// TIA Portal project "Assembler" (V16)
// Vorlageprojekt für das Buch mit Zielsystem S7-1200

(* hardware
DEVICE "S7-1200-Station_1"  S7-1200 Station
   slot 0: "Baugruppenträger_0"  Rack  V1.0
   slot 1: "PLC_1"  CPU 1211C DC/DC/DC  6ES7 211-1AE40-0XB0  V4.1
*)

// ===== PLC "PLC_1"  CPU 1211C DC/DC/DC =====

VAR_GLOBAL   // PLC tag table "Standard-Variablentabelle"
   "Start" AT %I0.0 : Bool;
   "Stop" AT %I0.1 : Bool;
   "Vision sensor (bool 0)" AT %I0.2 : Bool;
   "Vision sensor (bool 1)" AT %I0.3 : Bool;
   "pusher base (FL)" AT %I0.4 : Bool;
   "pusher base (BL)" AT %I0.5 : Bool;
   "pusher LID (FL)" AT %I0.6 : Bool;
   "pusher LID (BL)" AT %I0.7 : Bool;
   "DS BASE" AT %I1.0 : Bool;
   "DS LID" AT %I1.1 : Bool;
   "Base Clamped" AT %I1.2 : Bool;
   "LID Clamped" AT %I1.3 : Bool;
   "Item Leaving" AT %I1.4 : Bool;
   "Moving Z" AT %I1.5 : Bool;
   "Moving X" AT %I1.6 : Bool;
   "Item Detected" AT %I1.7 : Bool;
   "Sensor Base" AT %I2.0 : Bool;
   "Sensor LID" AT %I2.1 : Bool;
   "First Conv" AT %Q0.0 : Bool;
   "Main Conv" AT %Q0.1 : Bool;
   "Pusher Base" AT %Q0.2 : Bool;
   "Pusher LID" AT %Q0.3 : Bool;
   "Base Conv" AT %Q0.4 : Bool;
   "LID Conv" AT %Q0.5 : Bool;
   "Base Clamp" AT %Q0.6 : Bool;
   "LID Clamp" AT %Q0.7 : Bool;
   "Item Leave" AT %Q1.0 : Bool;
   "Move z" AT %Q1.1 : Bool;
   "Move x" AT %Q1.2 : Bool;
   "Grab" AT %Q1.3 : Bool;
   "X" AT %M0.0 : Bool;
   "X1" AT %M0.1 : Bool;
   "X2" AT %M0.2 : Bool;
   "X3" AT %M0.3 : Bool;
   "X4" AT %M0.4 : Bool;
   "X5" AT %M0.5 : Bool;
   "X6" AT %M0.6 : Bool;
   "X7" AT %M0.7 : Bool;
   "X8" AT %M1.0 : Bool;
   "X9" AT %M1.1 : Bool;
   "X10" AT %M1.2 : Bool;
   "X11" AT %M1.3 : Bool;
   "X12" AT %M1.4 : Bool;
   "X13" AT %M1.5 : Bool;
   "X14" AT %M1.6 : Bool;
   "X15" AT %M1.7 : Bool;
   "X16" AT %M2.0 : Bool;
   "X17" AT %M2.1 : Bool;
   "X18" AT %M2.2 : Bool;
   "X19" AT %M2.3 : Bool;
   "X20" AT %M2.4 : Bool;
   "X21" AT %M3.0 : Bool;
END_VAR

// folder: System blocks/Program resources

DATA_BLOCK "C1"   // DB1
{ S7_Optimized_Access := 'TRUE' }
AUTHOR : Simatic
FAMILY : IEC
NAME : CNTR
VERSION : 1.0
// stored: InstanceOfName IEC_COUNTER
"IEC_COUNTER"
BEGIN
END_DATA_BLOCK

DATA_BLOCK "T1"   // DB2
{ S7_Optimized_Access := 'TRUE' }
AUTHOR : Simatic
FAMILY : IEC
NAME : IEC_TMR
VERSION : 1.0
// stored: InstanceOfName IEC_TIMER
"IEC_TIMER"
BEGIN
END_DATA_BLOCK

// folder: (top level)

FUNCTION "MHJ-PLC-Lab-Function-S71200" : Void   // FC9000, SCL
{ S7_Optimized_Access := 'TRUE' }
VERSION : 0.1
   VAR_TEMP
      rdTimeReturn : Int;
      outputTime : DTL;
      SyncVal : Byte;
      forVal : Int;
      forVal_2 : Int;
      Value : Byte;
   END_VAR
   VAR CONSTANT
      CompVal : Byte := 16#34;
      Value_01 : Byte := 16#11;
      Value_01_DW : DWord := 16#A165_D992;
      Value_02_DW : DWord := 16#58BE_4401;
   END_VAR
BEGIN

   #Value:=PEEK(area := 16#82,
        dbNumber := 0,
        byteOffset := 511);
   #Value := #Value + 1;

   POKE(area := 16#82,
        dbNumber := 0,
        byteOffset := 511,
        value := #Value);

   POKE(area:=16#81,
        dbNumber:=0,
        byteOffset:=1016,
        value:=#Value_01_DW);
   POKE(area := 16#81,
        dbNumber := 0,
        byteOffset := 1020,
        value := #Value_02_DW);

   POKE(area := 16#81,
        dbNumber := 0,
        byteOffset := 511,
        value := B#16#00);

   FOR #forVal := 0 TO 120 DO
       FOR #forVal_2:=0 TO 10 DO
           #rdTimeReturn:=RD_SYS_T(#outputTime);
           #rdTimeReturn := WR_SYS_T(#outputTime);
           #rdTimeReturn := RD_SYS_T(#outputTime);
           #rdTimeReturn := WR_SYS_T(#outputTime);
       END_FOR;
       #SyncVal:= PEEK(area := 16#81,
                      dbNumber := 0,
                      byteOffset := 511);
       IF #SyncVal = #CompVal THEN
          GOTO M_1;
       END_IF;
   END_FOR;
   RETURN;

   M_1:
   POKE(area := 16#81,
        dbNumber := 0,
        byteOffset := 511,
        value := B#16#0);
END_FUNCTION

ORGANIZATION_BLOCK "Main"   // OB1, LAD, ProgramCycle
TITLE = "Main Program Sweep (Cycle)"
{ S7_Optimized_Access := 'TRUE' }
VERSION : 0.1
   VAR_INPUT
      Initial_Call : Bool;   // Initial call of this OB
      Remanence : Bool;   // =True, if remanent data are available
   END_VAR
   VAR_TEMP   // added for the SCL form of the ladder/FBD networks
      _w1 : Bool;
   END_VAR
BEGIN

REGION Network 1: Konnektierungsbaustein für PLC-Lab
   // Im Netzwerk 1 wird der Konnektierungsbaustein für PLC-Lab aufgerufen.
   // Dieser Aufruf darf nicht entfernt werden!
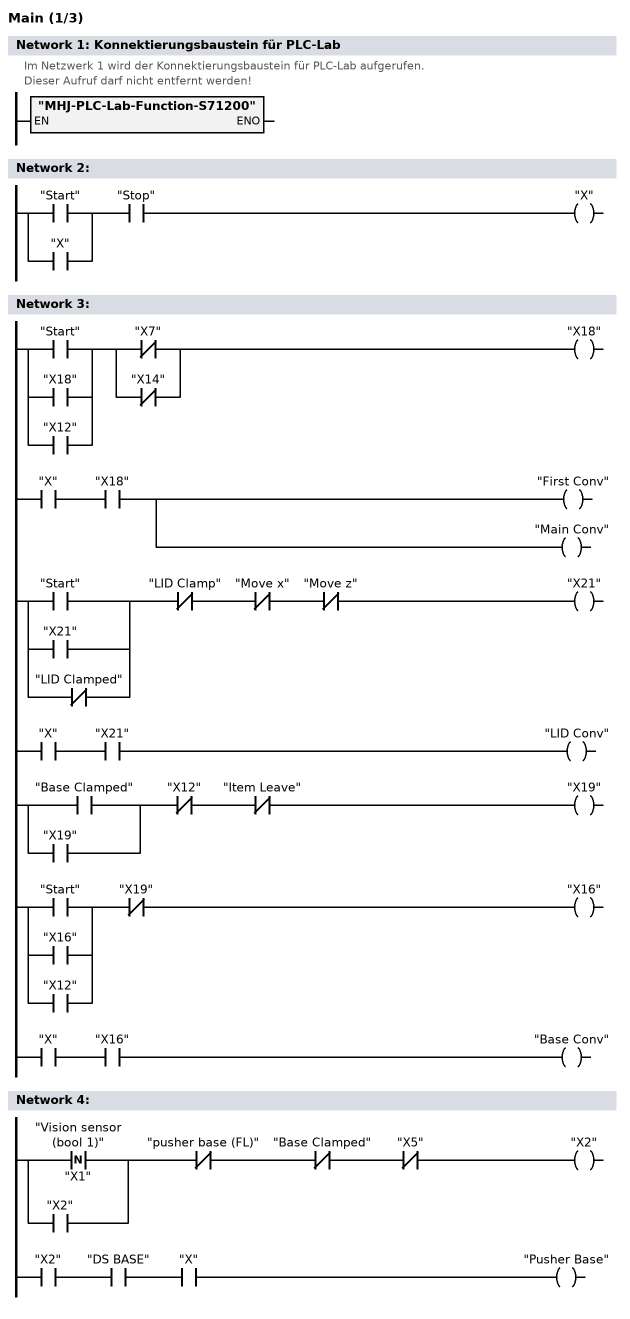
   RUNG wire#powerrail
      "MHJ-PLC-Lab-Function-S71200"()
   END_RUNG
   // the same network as SCL:
   "MHJ-PLC-Lab-Function-S71200"();
END_REGION

REGION Network 2
   RUNG wire#powerrail
      Contact( "Start" )
      wire#w1
      Contact( "Stop" )
      Coil( "X" )
   END_RUNG
   RUNG wire#powerrail
      Contact( "X" )
   END_RUNG wire#w1
   // the same network as SCL:
   "X" := ("Start" OR "X") AND "Stop";
END_REGION

REGION Network 3
   RUNG wire#powerrail
      Contact( "Start" )
      wire#w1
      I_Contact( "X7" )
      wire#w2
      Coil( "X18" )
   END_RUNG
   RUNG wire#powerrail
      Contact( "X18" )
   END_RUNG wire#w1
   RUNG wire#powerrail
      Contact( "X12" )
   END_RUNG wire#w1
   RUNG wire#w1
      I_Contact( "X14" )
   END_RUNG wire#w2
   RUNG wire#powerrail
      Contact( "X" )
      Contact( "X18" )
      wire#w3
      Coil( "First Conv" )
   END_RUNG
   RUNG wire#w3
      Coil( "Main Conv" )
   END_RUNG
   RUNG wire#powerrail
      Contact( "Start" )
      wire#w4
      I_Contact( "LID Clamp" )
      I_Contact( "Move x" )
      I_Contact( "Move z" )
      Coil( "X21" )
   END_RUNG
   RUNG wire#powerrail
      Contact( "X21" )
   END_RUNG wire#w4
   RUNG wire#powerrail
      I_Contact( "LID Clamped" )
   END_RUNG wire#w4
   RUNG wire#powerrail
      Contact( "X" )
      Contact( "X21" )
      Coil( "LID Conv" )
   END_RUNG
   RUNG wire#powerrail
      Contact( "Base Clamped" )
      wire#w5
      I_Contact( "X12" )
      I_Contact( "Item Leave" )
      Coil( "X19" )
   END_RUNG
   RUNG wire#powerrail
      Contact( "X19" )
   END_RUNG wire#w5
   RUNG wire#powerrail
      Contact( "Start" )
      wire#w6
      I_Contact( "X19" )
      Coil( "X16" )
   END_RUNG
   RUNG wire#powerrail
      Contact( "X16" )
   END_RUNG wire#w6
   RUNG wire#powerrail
      Contact( "X12" )
   END_RUNG wire#w6
   RUNG wire#powerrail
      Contact( "X" )
      Contact( "X16" )
      Coil( "Base Conv" )
   END_RUNG
   // the same network as SCL:
   "X18" := ("Start" OR "X18" OR "X12") AND (NOT "X7" OR NOT "X14");
   "First Conv" := "X" AND "X18";
   "Main Conv" := "First Conv";
   "X21" := ("Start" OR "X21" OR NOT "LID Clamped") AND NOT "LID Clamp" AND NOT "Move x" AND NOT "Move z";
   "LID Conv" := "X" AND "X21";
   "X19" := ("Base Clamped" OR "X19") AND NOT "X12" AND NOT "Item Leave";
   "X16" := ("Start" OR "X16" OR "X12") AND NOT "X19";
   "Base Conv" := "X" AND "X16";
END_REGION

REGION Network 4
   RUNG wire#powerrail
      N_Contact(operand := "Vision sensor (bool 1)", bit := "X1")
      wire#w1
      I_Contact( "pusher base (FL)" )
      I_Contact( "Base Clamped" )
      I_Contact( "X5" )
      Coil( "X2" )
   END_RUNG
   RUNG wire#powerrail
      Contact( "X2" )
   END_RUNG wire#w1
   RUNG wire#powerrail
      Contact( "X2" )
      Contact( "DS BASE" )
      Contact( "X" )
      Coil( "Pusher Base" )
   END_RUNG
   // the same network as SCL:
   #_w1 := NOT "Vision sensor (bool 1)" AND "X1";   // falling edge of "Vision sensor (bool 1)"
   "X1" := "Vision sensor (bool 1)";
   "X2" := (#_w1 OR "X2") AND NOT "pusher base (FL)" AND NOT "Base Clamped" AND NOT "X5";
   "Pusher Base" := "X2" AND "DS BASE" AND "X";
END_REGION

REGION Network 5
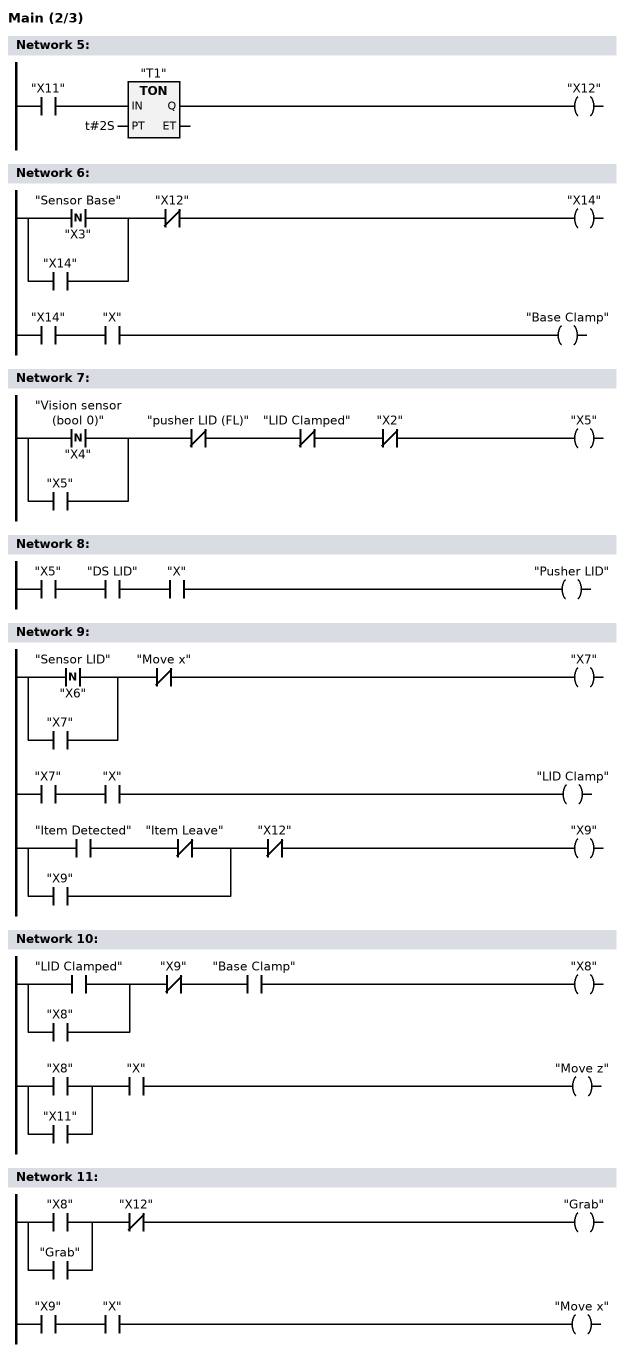
   "T1".TON(IN := "X11", PT := t#2S);
   "X12" := "T1".Q;
END_REGION

REGION Network 6
   RUNG wire#powerrail
      N_Contact(operand := "Sensor Base", bit := "X3")
      wire#w1
      I_Contact( "X12" )
      Coil( "X14" )
   END_RUNG
   RUNG wire#powerrail
      Contact( "X14" )
   END_RUNG wire#w1
   RUNG wire#powerrail
      Contact( "X14" )
      Contact( "X" )
      Coil( "Base Clamp" )
   END_RUNG
   // the same network as SCL:
   #_w1 := NOT "Sensor Base" AND "X3";   // falling edge of "Sensor Base"
   "X3" := "Sensor Base";
   "X14" := (#_w1 OR "X14") AND NOT "X12";
   "Base Clamp" := "X14" AND "X";
END_REGION

REGION Network 7
   RUNG wire#powerrail
      N_Contact(operand := "Vision sensor (bool 0)", bit := "X4")
      wire#w1
      I_Contact( "pusher LID (FL)" )
      I_Contact( "LID Clamped" )
      I_Contact( "X2" )
      Coil( "X5" )
   END_RUNG
   RUNG wire#powerrail
      Contact( "X5" )
   END_RUNG wire#w1
   // the same network as SCL:
   #_w1 := NOT "Vision sensor (bool 0)" AND "X4";   // falling edge of "Vision sensor (bool 0)"
   "X4" := "Vision sensor (bool 0)";
   "X5" := (#_w1 OR "X5") AND NOT "pusher LID (FL)" AND NOT "LID Clamped" AND NOT "X2";
END_REGION

REGION Network 8
   RUNG wire#powerrail
      Contact( "X5" )
      Contact( "DS LID" )
      Contact( "X" )
      Coil( "Pusher LID" )
   END_RUNG
   // the same network as SCL:
   "Pusher LID" := "X5" AND "DS LID" AND "X";
END_REGION

REGION Network 9
   RUNG wire#powerrail
      N_Contact(operand := "Sensor LID", bit := "X6")
      wire#w1
      I_Contact( "Move x" )
      Coil( "X7" )
   END_RUNG
   RUNG wire#powerrail
      Contact( "X7" )
   END_RUNG wire#w1
   RUNG wire#powerrail
      Contact( "X7" )
      Contact( "X" )
      Coil( "LID Clamp" )
   END_RUNG
   RUNG wire#powerrail
      Contact( "Item Detected" )
      I_Contact( "Item Leave" )
      wire#w2
      I_Contact( "X12" )
      Coil( "X9" )
   END_RUNG
   RUNG wire#powerrail
      Contact( "X9" )
   END_RUNG wire#w2
   // the same network as SCL:
   #_w1 := NOT "Sensor LID" AND "X6";   // falling edge of "Sensor LID"
   "X6" := "Sensor LID";
   "X7" := (#_w1 OR "X7") AND NOT "Move x";
   "LID Clamp" := "X7" AND "X";
   "X9" := (("Item Detected" AND NOT "Item Leave") OR "X9") AND NOT "X12";
END_REGION

REGION Network 10
   RUNG wire#powerrail
      Contact( "LID Clamped" )
      wire#w1
      I_Contact( "X9" )
      Contact( "Base Clamp" )
      Coil( "X8" )
   END_RUNG
   RUNG wire#powerrail
      Contact( "X8" )
   END_RUNG wire#w1
   RUNG wire#powerrail
      Contact( "X8" )
      wire#w2
      Contact( "X" )
      Coil( "Move z" )
   END_RUNG
   RUNG wire#powerrail
      Contact( "X11" )
   END_RUNG wire#w2
   // the same network as SCL:
   "X8" := ("LID Clamped" OR "X8") AND NOT "X9" AND "Base Clamp";
   "Move z" := ("X8" OR "X11") AND "X";
END_REGION

REGION Network 11
   RUNG wire#powerrail
      Contact( "X8" )
      wire#w1
      I_Contact( "X12" )
      Coil( "Grab" )
   END_RUNG
   RUNG wire#powerrail
      Contact( "Grab" )
   END_RUNG wire#w1
   RUNG wire#powerrail
      Contact( "X9" )
      Contact( "X" )
      Coil( "Move x" )
   END_RUNG
   // the same network as SCL:
   "Grab" := ("X8" OR "Grab") AND NOT "X12";
   "Move x" := "X9" AND "X";
END_REGION

REGION Network 12
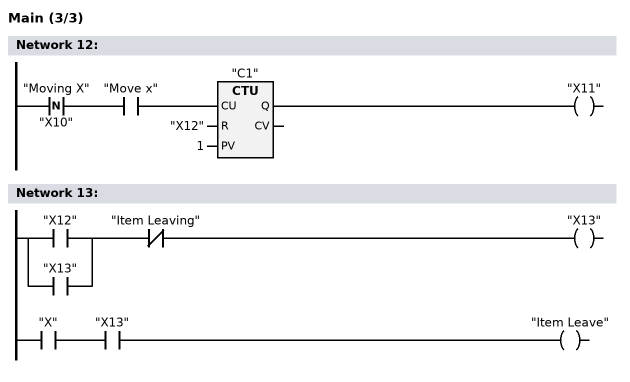
   #_w1 := NOT "Moving X" AND "X10";   // falling edge of "Moving X"
   "X10" := "Moving X";
   "C1".CTU(CU := #_w1 AND "Move x", R := "X12", PV := 1);
   "X11" := "C1".Q;
END_REGION

REGION Network 13
   RUNG wire#powerrail
      Contact( "X12" )
      wire#w1
      I_Contact( "Item Leaving" )
      Coil( "X13" )
   END_RUNG
   RUNG wire#powerrail
      Contact( "X13" )
   END_RUNG wire#w1
   RUNG wire#powerrail
      Contact( "X" )
      Contact( "X13" )
      Coil( "Item Leave" )
   END_RUNG
   // the same network as SCL:
   "X13" := ("X12" OR "X13") AND NOT "Item Leaving";
   "Item Leave" := "X" AND "X13";
END_REGION
END_ORGANIZATION_BLOCK